PROGRAM prgCS
VAR
	fbCSvirt	: FB_Light;
	bCSOn		: BOOL; //{#lynus.ag#()}
	bCSOff		: BOOL; //{#lynus.ag#()}
	bStateCS	: BOOL; //{#lynus.ag#()}
	lrCSpower	: LREAL; //{#lynus.ag#()}
END_VAR

fbCSvirt(bOn:=bCSOn, bOff:=bCSOff, bLight=>bStateCS);

IF bStateCS THEN
	lrCSpower := 11.02;
	ELSE
	lrCSpower := 0;
END_IF

END_PROGRAM

(* stored: Version 1.1.0.1, ProductVersion 3.1.4024.11
   POU prgCS: Id {c378a663-4727-4372-8964-04eba36a38f0}, SpecialFunc None *)
